ABB RobotStudio station: Solution2.rsstn

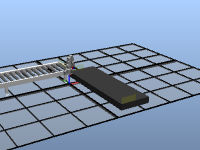
Station Solution2 (saved by RobotStudio 7.0.8504.151)
Controller Vinnie, task T_ROB1: task frame (RAPID world) sits at (0, 0, 400) mm in the station
Controller Vinnie
  mechanical unit ROB_1: IRB120_3_58__01, 6 joints, base frame (0, 0, 0) mm
Layout (positions relative to the parent item):
  - IRB120_3_58__01 [mechanism, from Robots\IRB120_3_58_G_01.rslib] at (0, 0, 400) mm; joint values [0, 0.1132, 1.2005, 0, 0.2571, 0] (rad or m)
  - Conveyor1 [smart component]
      signals: DI NewBox, DO BoxAtPos
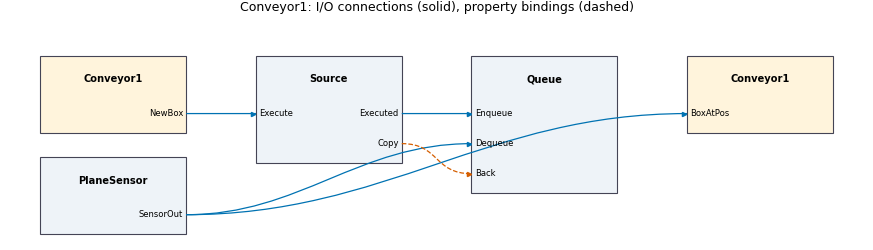
      connections:
        Conveyor1.NewBox -> Source.Execute
        Source.Executed -> Queue.Enqueue
        PlaneSensor.SensorOut -> Queue.Dequeue
        PlaneSensor.SensorOut -> Conveyor1.BoxAtPos
        Source.Copy => Queue.Back
    - 950_4000_h2 [part, from Equipment\Conveyor 950 4000 h2.rslib] at (-3846.63, 300, 0) mm
    - Source [smart component, from Components\Source.rslib]
        properties: Source=Part_1; Copy=(none); Parent=(none); Position=[0 0 0]; Orientation=[0 0 0]; Transient=false; PhysicsBehavior=0
    - Queue [smart component, from Components\Queue.rslib]
        properties: Back=(none); Front=(none); Queue={2cd56b75-4092-4768-a475-00f35c4dae8b};{e0dd32b4-5c51-4f0d-a48d-accb6fe5d5c2};{74c91f28-67c0-4405-bb46-46a2bebc9ae4};{4de452c9-d932-4406-abf8-51a8521f936e};{88fa9637-5f31-4297-a4ce-dfd895462f0a};{a1be2565-d57b-44ca-a3d4-488ed4227e35};{48cd2ff7-af39-436b-9b86-b527ae4f2f15};{69c433ef-7d00-473a-887e-093ac5fd6830}; NumberOfObjects=0
    - LinearMover [smart component, from Components\LinearMover.rslib]
        properties: Object=Queue; Direction=[1 0 0]; Speed=0.5; Reference=Global; ReferenceObject=(none)
    - PlaneSensor [smart component, from Components\PlaneSensor.rslib]
        properties: Origin=[0.162459 1.21 0.435]; Axis1=[0 -0.91 0]; Axis2=[0 0 0.2]; SensedPart=(none)
      - _sensorPart_ [part]
  - Part_1 [part]
  - Conveyor2 [smart component]
      signals: DI CakeReady, DO CakeStop, DO CakeDone, DI DecorationFinish
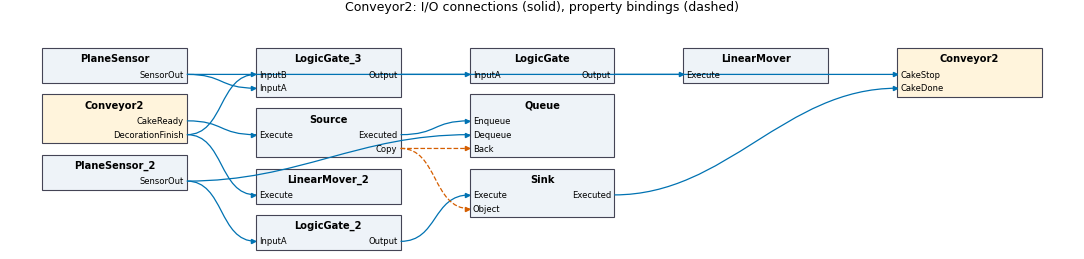
      connections:
        Source.Executed -> Queue.Enqueue
        PlaneSensor.SensorOut -> Conveyor2.CakeStop
        Sink.Executed -> Conveyor2.CakeDone
        LogicGate.Output -> LinearMover.Execute
        Conveyor2.CakeReady -> Source.Execute
        Conveyor2.DecorationFinish -> LinearMover_2.Execute
        PlaneSensor_2.SensorOut -> Queue.Dequeue
        PlaneSensor_2.SensorOut -> LogicGate_2.InputA
        LogicGate_2.Output -> Sink.Execute
        Conveyor2.DecorationFinish -> LogicGate_3.InputB
        PlaneSensor.SensorOut -> LogicGate_3.InputA
        LogicGate_3.Output -> LogicGate.InputA
        Source.Copy => Queue.Back
        Source.Copy => Sink.Object
    - Part_3 [part]
    - Source [smart component, from Components\Source.rslib]
        properties: Source=Part_4; Copy=(none); Parent=(none); Position=[0 0 0]; Orientation=[0 0 0]; Transient=false; PhysicsBehavior=0
    - LinearMover [smart component, from Components\LinearMover.rslib]
        properties: Object=Queue; Direction=[0 1 0]; Speed=0.5; Reference=Global; ReferenceObject=(none)
    - Queue [smart component, from Components\Queue.rslib]
        properties: Back=(none); Front=(none); Queue={c695aee4-bfaa-4f1e-a74f-64ccdeb8bb4b};{1af55ff9-90c2-46cc-8bb7-e61e5e7bc5cf};{b0d27663-1fba-4821-85d6-26657cc262f1};{f4cf88df-f486-4804-b77d-170edf7cc492};{4710dba7-5671-4460-a84a-d2ea9da19cfe};{420a59de-b4e8-43d9-a721-343f294f606b};{278b6554-ba95-48a2-b609-b906a8146629};{23ba5402-1793-4113-b4e2-e93ad0b6c6c6};{07cc2856-54ba-470d-9d90-e7ecf2db2aac};{00edcc47-4e0d-473d-8f5a-5610fa2a1b26};{5a767707-28a5-47a6-8cc2-16b9d7c295fa};{85b51734-0f60-45b7-9c93-7e9f9f0bd86e};{08f5d8c8-d7ee-4459-b28c-c8b0efa839b5}; NumberOfObjects=0
    - PlaneSensor [smart component, from Components\PlaneSensor.rslib]
        properties: Origin=[0.175 0.162 0.4]; Axis1=[0.5 0 0]; Axis2=[0 0 0.2]; SensedPart=(none)
      - _sensorPart_ [part]
    - Sink [smart component, from Components\Sink.rslib]
        properties: Object=(none)
    - PlaneSensor_2 [smart component, from Components\PlaneSensor.rslib]
        properties: Origin=[0.130644 -3 0.4]; Axis1=[0.5 0 0]; Axis2=[0 0 0.2]; SensedPart=(none)
      - _sensorPart_ [part]
    - LogicGate [smart component, from Components\LogicGate.rslib]
        properties: Operator=NOT; Delay=0
    - LinearMover_2 [smart component, from Components\LinearMover.rslib]
        properties: Object=Queue; Direction=[0 -1 0]; Speed=0.5; Reference=Global; ReferenceObject=(none)
    - LogicGate_2 [smart component, from Components\LogicGate.rslib]
        properties: Operator=AND; Delay=1
    - LogicGate_3 [smart component, from Components\LogicGate.rslib]
        properties: Operator=OR; Delay=0
  - Part_4 [part] at (0, 50, 0) mm
Station signals: DI Start
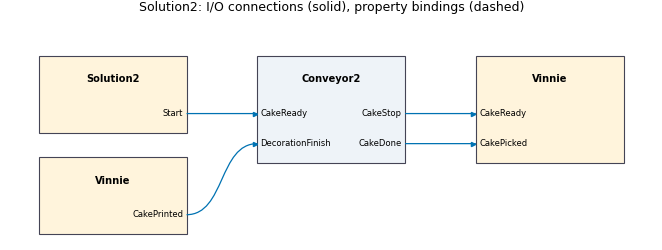
Station logic (signal -> signal, property => property):
  Conveyor2.CakeStop -> Vinnie.CakeReady
  Solution2.Start -> Conveyor2.CakeReady
  Conveyor2.CakeDone -> Vinnie.CakePicked
  Vinnie.CakePrinted -> Conveyor2.DecorationFinish
